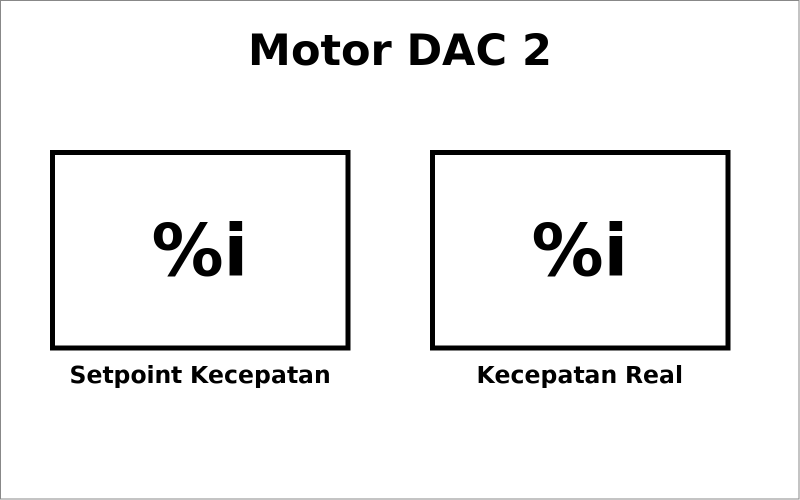
VISUALIZATION Screen_2_Sub_6  // 800x500
    Label (0,0 800x100), "Motor DAC 2"
    Rectangle (50,150 300x200), "%i", text variable: GVL.HMI_Motor_DAC_2_Input
        OnMouseClick: write GVL.HMI_Motor_DAC_2_Input via VisuDialogs.Numpad
    Label (50,350 300x50), "Setpoint Kecepatan"
    Label (430,350 300x50), "Kecepatan Real"
    Rectangle (430,150 300x200), "%i", text variable: GVL.HMI_Motor_DAC_2_Real
END_VISUALIZATION

(* stored: Version 1.1.0.1, ProductVersion 3.1.4024.12
   Visu Screen_2_Sub_6: Id {a4444a3b-ffbb-40ae-bf4a-86638486fe5c} *)
